FUNCTION_BLOCK FB_MotionAxisNC IMPLEMENTS I_MotionAxis
VAR
    AxisReference : REFERENCE TO AXIS_REF;

    bCommandedReset : BOOL;
    fbMcReset : MC_Reset;
    bMostRecentResetDone : BOOL;

    fbMcPower : MC_Power;

    bCommandedHome : BOOL;
    fbMcHome : MC_Home;
    bMostRecentHomeDone : BOOL;

    bCommandedHalt : BOOL;
    fbMcHalt : MC_Halt;
    bMostRecentHaltDone : BOOL;

    bCommandedMoveAbsolute : BOOL;
    fbMcMoveAbsolute : MC_MoveAbsolute;
    bMostRecentMoveAbsoluteDone : BOOL;

    bCommandedGearIn : BOOL;
    fbMcGearIn : MC_GearIn;

    bCommandedGearOut : BOOL;
    fbMcGearOut : MC_GearIn;
END_VAR


IF THIS^.AxisReference.NcToPlc.AxisId = 0 THEN
    RETURN;
END_IF

THIS^.AxisReference.ReadStatus();

THIS^.fbMcReset(
    Axis := THIS^.AxisReference,
    Execute := THIS^.bCommandedReset
);
THIS^.bCommandedReset := FALSE;

IF THIS^.fbMcReset.Done THEN
    THIS^.bMostRecentResetDone := TRUE;
END_IF

THIS^.fbMcPower(
    Axis := THIS^.AxisReference
);

THIS^.fbMcHome(
    Axis := THIS^.AxisReference,
    Execute := THIS^.bCommandedHalt
);
THIS^.bCommandedHome := FALSE;

IF THIS^.fbMcHome.Done THEN
    THIS^.bMostRecentHomeDone := TRUE;
END_IF

THIS^.fbMcHalt(
    Axis := THIS^.AxisReference,
    Execute := THIS^.bCommandedHalt
);
THIS^.bCommandedHalt := FALSE;

IF THIS^.fbMcHalt.Done THEN
    THIS^.bMostRecentHaltDone := TRUE;
END_IF

THIS^.fbMcMoveAbsolute(
    Axis := THIS^.AxisReference,
    Execute := THIS^.bCommandedMoveAbsolute
);
THIS^.bCommandedMoveAbsolute := FALSE;

IF THIS^.fbMcMoveAbsolute.Done THEN
    THIS^.bMostRecentMoveAbsoluteDone := TRUE;
END_IF

{warning 'Add method implementation '}
METHOD CalibrateEncValue
END_METHOD

{warning 'Add method implementation '}
METHOD EncSaveRestore
END_METHOD

{warning 'Add property implementation'}
PROPERTY Error : BOOL
GET
END_GET
END_PROPERTY

{warning 'Add property implementation'}
PROPERTY ErrorID : BOOL
GET
END_GET
END_PROPERTY


METHOD FB_Init: BOOL
VAR_INPUT
    bInitRetains: BOOL; // TRUE: the retain variables are initialized (reset warm / reset cold)
    bInCopyCode: BOOL;  // TRUE: the instance will be copied to the copy code afterward (online change)

    AxisReference : REFERENCE TO AXIS_REF;
END_VAR

THIS^.AxisReference REF= AxisReference;
END_METHOD

{warning 'Add method implementation '}
METHOD GearIn
END_METHOD

{warning 'Add method implementation '}
METHOD GearOut
END_METHOD


METHOD GetAxisRef : REFERENCE TO AXIS_REF

GetAxisRef REF= THIS^.AxisReference;
END_METHOD


METHOD GetPowerOverride : LREAL

GetPowerOverride := TO_LREAL(THIS^.AxisReference.PlcToNc.Override) / 10000.0;
END_METHOD


METHOD Halt
VAR_INPUT
    Deceleration	: LREAL := 0.0;
    Jerk	: LREAL := 0.0;
    BufferMode	: MC_BufferMode := .MC_BufferMode.MC_Aborting;
END_VAR
VAR_OUTPUT
    Done	: BOOL;
    Busy	: BOOL;
    Active	: BOOL;
    CommandAborted	: BOOL;
    Error	: BOOL;
    ErrorID	: UDINT;
    ErrorStr	: T_MaxString;
END_VAR

bMostRecentHaltDone := FALSE;

IF NOT HaltBusy THEN
    bCommandedHalt := TRUE;
END_IF

THIS^.fbMcHalt(
    Axis := THIS^.AxisReference,
    Deceleration := Deceleration,
    Jerk := Jerk,
    BufferMode := BufferMode,
    Done => Done,
    Busy => Busy,
    Active => Active,
    CommandAborted => CommandAborted,
    Error => Error,
    ErrorID => ErrorID
);

ErrorStr := '';
END_METHOD


PROPERTY HaltBusy : BOOL
GET

HaltBusy := THIS^.fbMcHalt.Busy;
END_GET
END_PROPERTY


PROPERTY HaltDone : BOOL
GET

HaltDone := THIS^.fbMcHalt.Done OR THIS^.bMostRecentHaltDone;
END_GET
END_PROPERTY


PROPERTY HaltError : BOOL
GET

HaltError := THIS^.fbMcHalt.Error;
END_GET
END_PROPERTY


PROPERTY HaltErrorID : UDINT
GET

HaltErrorID := THIS^.fbMcHalt.ErrorID;
END_GET
END_PROPERTY


METHOD Home
VAR_INPUT
    Position : LREAL := DEFAULT_HOME_POSITION;
    HomingMode : MC_HomingMode := MC_DefaultHoming;
END_VAR
VAR_OUTPUT
    Done	: BOOL;
    Busy	: BOOL;
    Active	: BOOL;
    CommandAborted	: BOOL;
    Error	: BOOL;
    ErrorID	: UDINT;
    ErrorStr	: T_MaxString;
END_VAR

bMostRecentHomeDone := FALSE;

IF NOT HomeBusy THEN
    bCommandedHome := TRUE;
END_IF

THIS^.fbMcHome(
    Axis := THIS^.AxisReference,
    HomingMode := HomingMode,
    Done => Done,
    Busy => Busy,
    Active => Active,
    CommandAborted => CommandAborted,
    Error => Error,
    ErrorID => ErrorID
);

ErrorStr := '';
END_METHOD


PROPERTY HomeBusy : BOOL
GET

HomeBusy := THIS^.fbMcHome.Busy;
END_GET
END_PROPERTY


PROPERTY HomeDone : BOOL
GET

HomeDone := THIS^.fbMcHome.Done;
END_GET
END_PROPERTY


PROPERTY MeasuredAcceleration : LREAL
GET

MeasuredAcceleration := THIS^.AxisReference.NcToPlc.ActAcc;
END_GET
END_PROPERTY


PROPERTY MeasuredPosition : LREAL
GET

MeasuredPosition := THIS^.AxisReference.NcToPlc.ActPos;
END_GET
END_PROPERTY


PROPERTY MeasuredVelocity : LREAL
GET

MeasuredVelocity := THIS^.AxisReference.NcToPlc.ActVelo;
END_GET
END_PROPERTY


METHOD MoveAbsolute
VAR_INPUT
    Position	: LREAL;
    Velocity	: LREAL;
    Acceleration	: LREAL := 0.0;
    Deceleration	: LREAL := 0.0;
    Jerk	: LREAL := 0.0;
    BufferMode	: MC_BufferMode := .MC_BufferMode.MC_Aborting;
END_VAR
VAR_OUTPUT
    Done	: BOOL;
    Busy	: BOOL;
    Active	: BOOL;
    CommandAborted	: BOOL;
    Error	: BOOL;
    ErrorID	: UDINT;
    ErrorStr	: T_MaxString;
END_VAR

bMostRecentMoveAbsoluteDone := FALSE;

IF NOT MoveAbsoluteBusy THEN
    bCommandedMoveAbsolute := TRUE;
END_IF

THIS^.fbMcMoveAbsolute(
    Axis := THIS^.AxisReference,
    Position := Position,
    Velocity := Velocity,
    Acceleration := Acceleration,
    Deceleration := Deceleration,
    Jerk := Jerk,
    BufferMode := BufferMode,
    Done => Done,
    Busy => Busy,
    Active => Active,
    CommandAborted => CommandAborted,
    Error => Error,
    ErrorID => ErrorID
);

ErrorStr := '';
END_METHOD


PROPERTY MoveAbsoluteBusy : BOOL
GET

MoveAbsoluteBusy := THIS^.fbMcMoveAbsolute.Busy;
END_GET
END_PROPERTY


PROPERTY MoveAbsoluteDone : BOOL
GET

MoveAbsoluteDone := THIS^.fbMcMoveAbsolute.Done OR THIS^.bMostRecentMoveAbsoluteDone;
END_GET
END_PROPERTY


PROPERTY MoveAbsoluteError : BOOL
GET

MoveAbsoluteError := THIS^.fbMcMoveAbsolute.Error;
END_GET
END_PROPERTY


PROPERTY MoveAbsoluteErrorID : UDINT
GET

MoveAbsoluteErrorID := THIS^.fbMcMoveAbsolute.ErrorID;
END_GET
END_PROPERTY


PROPERTY MoveAbsoluteTargetAcceleration : LREAL
GET

MoveAbsoluteTargetAcceleration := THIS^.fbMcMoveAbsolute.Acceleration;
END_GET
END_PROPERTY


PROPERTY MoveAbsoluteTargetDeceleration : LREAL
GET

MoveAbsoluteTargetDeceleration := THIS^.fbMcMoveAbsolute.Deceleration;
END_GET
END_PROPERTY


PROPERTY MoveAbsoluteTargetJerk : LREAL
GET

MoveAbsoluteTargetJerk := THIS^.fbMcMoveAbsolute.Jerk;
END_GET
END_PROPERTY


PROPERTY MoveAbsoluteTargetPosition : LREAL
GET

MoveAbsoluteTargetPosition := THIS^.fbMcMoveAbsolute.Position;
END_GET
END_PROPERTY


PROPERTY MoveAbsoluteTargetVelocity : LREAL
GET

MoveAbsoluteTargetVelocity := THIS^.fbMcMoveAbsolute.Velocity;
END_GET
END_PROPERTY


PROPERTY MoveBusy : BOOL
GET

MoveBusy := HaltBusy OR HomeBusy OR MoveAbsoluteBusy;
END_GET
END_PROPERTY


PROPERTY MoveDone : BOOL
GET

MoveDone := HaltDone AND HomeDone AND MoveAbsoluteDone;
END_GET
END_PROPERTY


PROPERTY NegativeMotionIsEnabled : BOOL
GET

NegativeMotionIsEnabled := THIS^.AxisReference.PlcToNc.ControlDWord.2;
END_GET
END_PROPERTY


PROPERTY PositiveMotionIsEnabled : BOOL
GET

PositiveMotionIsEnabled := THIS^.AxisReference.PlcToNc.ControlDWord.1;
END_GET
END_PROPERTY


METHOD Power
VAR_INPUT
    Enable	: BOOL;
    Enable_Positive	: BOOL;
    Enable_Negative	: BOOL;
    (* in percent from 0 to 100 *)
    Override	: LREAL := 100.0;
    BufferMode	: MC_BufferMode := .MC_BufferMode.MC_Aborting;
END_VAR
VAR_OUTPUT
    Status	: BOOL;
    Busy	: BOOL;
    Active	: BOOL;
    Error	: BOOL;
    ErrorID	: UDINT;
    ErrorStr	: T_MaxString;
END_VAR

THIS^.fbMcPower(
    Axis := THIS^.AxisReference,
    Enable := Enable,
    Enable_Positive := Enable_Positive,
    Enable_Negative := Enable_Negative,
    Override := Override,
    BufferMode := BufferMode,
    Status => Status,
    Busy => Busy,
    Active => Active,
    Error => Error,
    ErrorID => ErrorID
);

ErrorStr := '';
END_METHOD


PROPERTY PowerError : BOOL
GET

PowerError := THIS^.fbMcPower.Error;
END_GET
END_PROPERTY


PROPERTY PowerErrorID : UDINT
GET

PowerErrorID := THIS^.fbMcPower.ErrorID;
END_GET
END_PROPERTY


PROPERTY PowerIsEnabled : BOOL
GET

PowerIsEnabled := THIS^.AxisReference.PlcToNc.ControlDWord.0;
END_GET
END_PROPERTY


PROPERTY PowerOverride : LREAL
GET

PowerOverride := GetPowerOverride();
END_GET
END_PROPERTY

{warning 'Add property implementation'}
PROPERTY PowerStatus : BOOL
GET

PowerStatus := THIS^.fbMcPower.Status;
END_GET
END_PROPERTY


METHOD Reset
VAR_OUTPUT
    Done	: BOOL;
    Busy	: BOOL;
    Error	: BOOL;
    ErrorID	: UDINT;
    ErrorStr	: T_MaxString;
END_VAR

bMostRecentResetDone := FALSE;

IF NOT ResetBusy THEN
    bCommandedReset := TRUE;
END_IF

THIS^.fbMcReset(
    Axis := THIS^.AxisReference,
    Done => Done,
    Busy => Busy,
    Error => Error,
    ErrorID => ErrorID,
);

ErrorStr := '';
END_METHOD


PROPERTY ResetBusy : BOOL
GET

ResetBusy := fbMcReset.Busy;
END_GET
END_PROPERTY


PROPERTY ResetDone : BOOL
GET

ResetDone := fbMcReset.Done;
END_GET
END_PROPERTY


PROPERTY ResetError : BOOL
GET

ResetError := fbMcReset.Error;
END_GET
END_PROPERTY


PROPERTY ResetErrorID : UDINT
GET

ResetErrorID := fbMcReset.ErrorID;
END_GET
END_PROPERTY


PROPERTY SetpointAcceleration : LREAL
GET

SetpointAcceleration := THIS^.AxisReference.NcToPlc.SetAcc;
END_GET
END_PROPERTY


PROPERTY SetpointJerk : LREAL
GET

SetpointJerk := THIS^.AxisReference.NcToPlc.SetJerk;
END_GET
END_PROPERTY


PROPERTY SetpointPosition : LREAL
GET

SetpointPosition := THIS^.AxisReference.NcToPlc.SetPos;
END_GET
END_PROPERTY


PROPERTY SetpointVelocity : LREAL
GET

SetpointVelocity := THIS^.AxisReference.NcToPlc.SetVelo;
END_GET
END_PROPERTY


METHOD SetPowerOverride
VAR_INPUT
    (* in percent from 0 to 100 *)
    Override	: LREAL;
END_VAR
VAR_OUTPUT
    Status	: BOOL;
    Busy	: BOOL;
    Active	: BOOL;
    Error	: BOOL;
    ErrorID	: UDINT;
    ErrorStr	: T_MaxString;
END_VAR

THIS^.fbMcPower(
    Axis := THIS^.AxisReference,
    Override := Override,
    Status => Status,
    Busy => Busy,
    Error => Error,
    ErrorID => ErrorID
);

ErrorStr := '';
END_METHOD

END_FUNCTION_BLOCK

(* stored: Version 1.1.0.1
   POU FB_MotionAxisNC: Id {96c72d7b-b1c4-4404-8b3a-a6e3d3eb1591}, SpecialFunc None
   Method CalibrateEncValue: Id {8ca97371-35e0-46e6-a9b7-7594354d8321}
   Method EncSaveRestore: Id {8ec82e12-941b-4df9-82d5-1d59ec9e96c0}
   Property Error: Id {0c9211cb-8ee9-464c-b55f-c17c79529917}
   Get Get: Id {7a94fb96-1282-4daa-b23d-9fab6525d751}
   Property ErrorID: Id {c0d033e6-fac9-42c2-a264-abf68bb57265}
   Get Get: Id {9472c55f-1675-43f9-806d-705fa9e88197}
   Method FB_Init: Id {bac111e8-1d7d-4fd4-a857-315a7e200ade}
   Method GearIn: Id {81dd8934-e3b1-4bec-b385-b138854f2123}
   Method GearOut: Id {c0b5a9df-5b8c-4db7-b16f-e5469da2a0df}
   Method GetAxisRef: Id {10d35074-4fd8-4e8b-9069-7e7f7f6a8421}
   Method GetPowerOverride: Id {2fddb9b6-12af-4c75-abad-4606be559da5}
   Method Halt: Id {da8196f8-e196-40ef-8a6e-bc6c7e6fbe2c}
   Property HaltBusy: Id {62ce211c-1234-4d0f-9c45-3c9cbe5e6003}
   Get Get: Id {4d24f738-494e-42ef-806b-8e70966de25f}
   Property HaltDone: Id {afe8d5cb-1d99-4048-9590-1a3920abe255}
   Get Get: Id {279f66bd-d06d-497a-84d9-c98540a0a364}
   Property HaltError: Id {4fadf73c-6771-4e18-b894-7ee5fbcf3779}
   Get Get: Id {c8129817-b180-45e4-b0a3-0a87c73f2d6d}
   Property HaltErrorID: Id {e98ef460-4348-454f-b52b-d723ef425d06}
   Get Get: Id {ece9775c-37a3-409f-ac65-cc8300570621}
   Method Home: Id {3bf2b3c3-9806-4f9f-aabb-f8586cc84efd}
   Property HomeBusy: Id {32c75310-58cd-47ec-b886-9ed752d7daf6}
   Get Get: Id {2d4452bc-ce84-46b2-a29b-c812f3643a1b}
   Property HomeDone: Id {66337a40-4a3c-4d92-bf24-6ddce48c0d91}
   Get Get: Id {606d437f-f82a-48fa-a81f-ec0d3aeec3ea}
   Property MeasuredAcceleration: Id {5fe95eb9-f25b-4824-9824-5ac23d2a939c}
   Get Get: Id {23d94457-e3d0-4862-bb28-c606a9b4e040}
   Property MeasuredPosition: Id {7aa4d620-42e9-46cf-a9e5-456428f89f41}
   Get Get: Id {0d0e6235-a791-4a18-ada6-053279f8e06c}
   Property MeasuredVelocity: Id {0d279219-54d3-43ff-9b4b-f55219fbc583}
   Get Get: Id {cbc9afab-0dce-417d-98bb-6eba68255088}
   Method MoveAbsolute: Id {67ccbbec-9b62-4af8-991b-52183ec6ce81}
   Property MoveAbsoluteBusy: Id {288161c6-71f9-4747-b207-784d14c7bb18}
   Get Get: Id {3410c6e1-ac91-46f6-add0-5e20046ced02}
   Property MoveAbsoluteDone: Id {4d9ec560-84bb-4ad6-9bf8-2100ac85ae39}
   Get Get: Id {eeee28e3-e5e6-475f-8f8b-a47b931517b2}
   Property MoveAbsoluteError: Id {0766c13f-dc50-4333-bdc9-27c1e8041e87}
   Get Get: Id {8e7c632e-6fff-431b-916a-d0bdc09c0394}
   Property MoveAbsoluteErrorID: Id {b7d1089e-1fca-460c-affe-a919a8311e55}
   Get Get: Id {5a444f3c-7c5d-40c7-ab2f-4666c84acbf7}
   Property MoveAbsoluteTargetAcceleration: Id {b0b8848e-299c-4ac6-85e8-10a4ed01d5b7}
   Get Get: Id {d782b91f-4097-4c28-b1a0-476041221974}
   Property MoveAbsoluteTargetDeceleration: Id {d5cb2321-79f3-4a78-924d-cf7595a947a8}
   Get Get: Id {6347c979-69fb-4625-8e3a-83400c69f397}
   Property MoveAbsoluteTargetJerk: Id {d9e05547-bba4-48a7-8e40-9c9718e2c053}
   Get Get: Id {8cde4a87-0890-4704-858e-0bed53aa2ff1}
   Property MoveAbsoluteTargetPosition: Id {db064498-2489-480c-8e8e-78251f5163d9}
   Get Get: Id {66ace398-70a2-4f96-87a5-784be92a971b}
   Property MoveAbsoluteTargetVelocity: Id {9ea06b23-062e-4e44-8536-72e608242537}
   Get Get: Id {b8a77f9a-bce3-409c-94d7-6127f641560f}
   Property MoveBusy: Id {aa1fb74c-1b50-4d51-8133-f13677216f50}
   Get Get: Id {3f11b9d7-655b-4ffe-abb7-eb8785d065bb}
   Property MoveDone: Id {e8da8efd-6713-4af4-a268-4d471d1e4497}
   Get Get: Id {6626854f-9461-4468-b96d-d25753f7b563}
   Property NegativeMotionIsEnabled: Id {35f5fd1a-af9f-48de-a9a3-ceb0e5406d38}
   Get Get: Id {fdda8cee-eef0-4d7f-8246-ea80f7ed0cae}
   Property PositiveMotionIsEnabled: Id {b1dc9334-1a69-4a47-ac75-8b8537dab0f0}
   Get Get: Id {27b35a92-fadb-4186-beb3-fe81d361a982}
   Method Power: Id {7c7f29eb-e69b-4866-a660-b5ec6c5a2421}
   Property PowerError: Id {a70a8f77-c387-45c0-a6a0-61fdeeaf7b69}
   Get Get: Id {d4386570-b633-408e-98f8-6063019e80e0}
   Property PowerErrorID: Id {fd7023c0-42e0-4958-b26d-25c003f8561c}
   Get Get: Id {8b2eae2f-0307-49a4-be29-c82a9978badc}
   Property PowerIsEnabled: Id {c5a19d8f-caa2-4df5-96f4-51ee6bc45944}
   Get Get: Id {d676e7c2-a963-498d-9de0-a55ac4f5e643}
   Property PowerOverride: Id {b50cb53b-78fc-41e3-9673-a36e3576e097}
   Get Get: Id {f8f17b65-52cb-4a25-9375-684bbd81f38b}
   Property PowerStatus: Id {d7ea7765-c440-4a7f-a984-6a3660dc9cb4}
   Get Get: Id {df6a4db9-be9b-44ff-a98e-b92944e682f8}
   Method Reset: Id {59ae1b7c-b5c5-42d3-954c-92f328e97d5f}
   Property ResetBusy: Id {2483eb0f-cd72-4e71-af17-0e53aa87faa8}
   Get Get: Id {74136afb-5824-4ead-b660-ab776cd949e5}
   Property ResetDone: Id {7d8fe4ef-bebc-41ad-ab5f-d8228e86dc97}
   Get Get: Id {99dd92af-06a9-40c0-9b61-ae55954b6d47}
   Property ResetError: Id {f26378fe-a781-4736-81af-8e55422df90a}
   Get Get: Id {59278bd6-2d98-4f6b-85b9-4ab95760783b}
   Property ResetErrorID: Id {b2c9c20f-1158-4dc5-a450-388c6f5be22e}
   Get Get: Id {0cc9c431-57e0-4475-97c3-74c073ceba1c}
   Property SetpointAcceleration: Id {0600d181-611e-4f4a-a8c1-ffc8acf60510}
   Get Get: Id {fb3abcd8-31bb-4455-a4db-125f47f14dfe}
   Property SetpointJerk: Id {ce1a269a-6507-4562-8a86-5bb71ff9b1b9}
   Get Get: Id {f71dc33e-887c-42e9-ac9b-3bcf07ff102e}
   Property SetpointPosition: Id {23952526-91d2-43d8-a75d-e10f448d76c7}
   Get Get: Id {f87853b8-9b08-4b7c-a83b-545cc754fb92}
   Property SetpointVelocity: Id {919c9874-73ab-4280-88de-6535d4a15bc0}
   Get Get: Id {26064423-fa6d-488a-ba6e-c34582673e26}
   Method SetPowerOverride: Id {76dd2720-0006-4788-b748-58af6a96df71} *)
